RoboDK station: kr30 cnc 081119 3.rdk

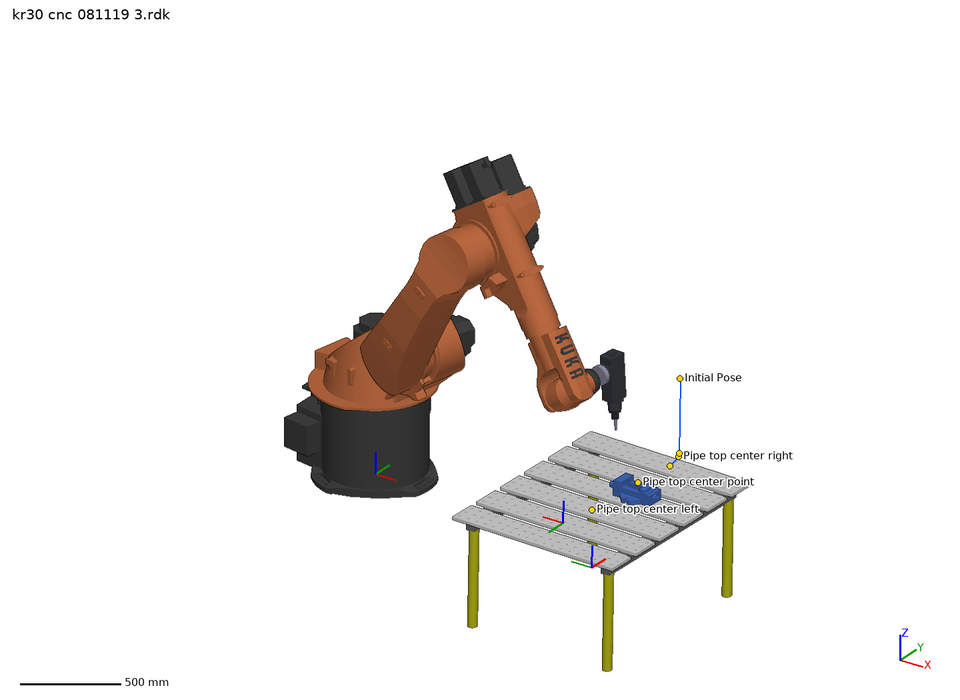
[picture v0: the station drawn from its stored meshes, robots at their saved joint values, targets as dots, program paths as lines]
Station kr30 cnc 081119 3. Poses are relative to the parent item; angles as X-Y-Z fixed-axis rotations.
  - frame GIGASHEEN Base at (0, 0, 0) mm
    - robot GIGASHEEN (model KUKA KR 30 HA): 6 axes, payload 30 kg, reach 2033 mm, repeatability 0.05 mm, weight 665 kg
        modified DH rows (alpha deg, a mm, theta deg, d mm): 0, 0, 0, 815; -90, 350, 0, 0; 0, 850, -90, 0; -90, 145, 0, 820; 90, 0, 0, 0; -90, 0, 180, 170
        joint limits [-185, -135, -120, -350, -119, -350] to [185, 35, 158, 350, 119, 350]; home [0, -90, 90, 0, 0, 0]; saved at [10.82, -58.087, 115.091, 93.153, -93.957, -30.819]
      - tool 1/8" Round Nose, TCP at (245.54, -0.16, 160.54) mm, rotated rx 0 ry 90 rz 0 deg, size 415.8 x 102 x 153.6 mm, geometry from GIGASHEEN
  - frame Table at (1949.02, -919.97, 396.91) mm, rotated rx 0.87 ry 0.27 rz 90 deg
    - frame Frame 4 at (440, 480, -70) mm, rotated rx 0 ry 0 rz 90 deg
      - object Table at (0, -330, 0) mm, rotated rx 0 ry 0 rz 90 deg, size 1193.8 x 965.2 x 609.6 mm, geometry from welding_table.sld
      - object Assembly at (-280, -390, 40) mm, size 290 x 180.6 x 89.2 mm, geometry from Assembly.igs
      - target Pipe top center left (joint target) at (-172.21, -0.54, 122.71) mm, rotated rx -178.45 ry -1.01 rz -2.71 deg; joints [18.81, -49.92, 112.957, 18.225, -62.324, -6.296] of GIGASHEEN
      - target Pipe top center right (joint target) at (-176.14, -744.37, 123.67) mm, rotated rx -177.29 ry -1.54 rz 86.1 deg; joints [1.888, -40.092, 92.828, 89.55, -87.31, -35.426] of GIGASHEEN
      - target Pipe top center point (joint target) at (-177.32, -391.58, 123.25) mm, rotated rx -177.29 ry -1.54 rz 86.1 deg; joints [14.13, -37.547, 87.475, 99.077, -95.14, -37.636] of GIGASHEEN
      - target Initial Pose (joint target) at (-176.14, -744.37, 553.67) mm, rotated rx -177.29 ry -1.54 rz 86.1 deg; joints [1.92, -52.358, 87.431, 90.405, -87.326, -53.108] of GIGASHEEN
      - target First slot (joint target) at (-176.14, -668.17, 105) mm, rotated rx -177.29 ry -1.54 rz 86.1 deg; joints [4.695, -34.361, 91.231, 91.707, -88.884, -31.273] of GIGASHEEN
      - target First slot retract (joint target) at (-176.14, -744.37, 143.67) mm, rotated rx -177.29 ry -1.54 rz 86.1 deg; joints [1.996, -36.427, 91.974, 89.507, -87.397, -32.612] of GIGASHEEN
  - program Prog1 (8 instructions, listed below)
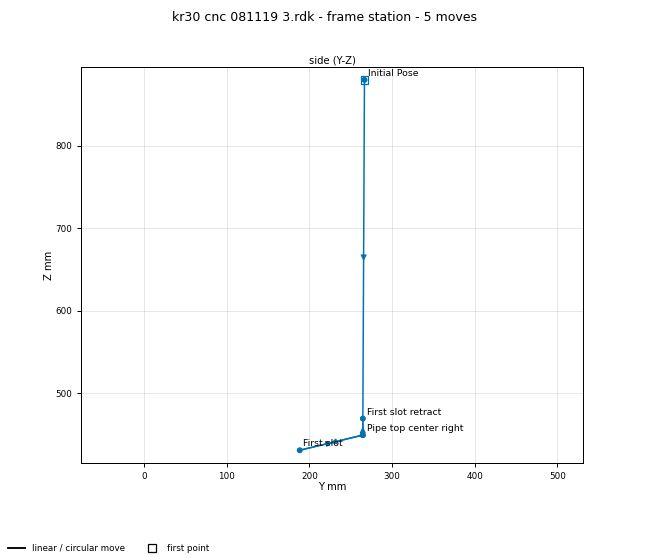
[picture p0: tool path of kr30 cnc 081119 3.rdk in frame station, 5 of 5 moves have a stored position in this frame; points joined in program order, loops and branches not executed]

--- program Prog1 (robot GIGASHEEN) ---
  Set Ref.: Frame 4
  Set Tool: 1/2" End Mill TCP -> 1/8" Round Nose
  MoveJ (Target 4) -> target Initial Pose
  MoveL (Pipe top center right)
  Set speed (2.0 mm/s)
  MoveL (Target 5) -> target First slot
  MoveL (Pipe top center right)
  MoveL (Target 6) -> target First slot retract
